KUKA KRL program: end_weld_respot.src

&ACCESS RVO3
&REL 149
&COMMENT end_weld_RESPOT
&PARAM DISKPATH = KRC:\R1\Program\SubRotinas
DEF end_weld_RESPOT( )
;
; FIM DO PROCESSO DE SOLDAGEM
;FOLD PULSE 3333 'R2 trabalho concluído-845' State=TRUE Time=3 sec;%{PE}%R 8.2.20,%MKUKATPBASIS,%COUT,%VPULSE,%P 2:3333, 3:R2 trabalho concluído-845, 5:TRUE, 6:, 8:3
PULSE($OUT[3333], TRUE,3)
;ENDFOLD
;
END
